Universal Robots PolyScope program: mixerHome.urp

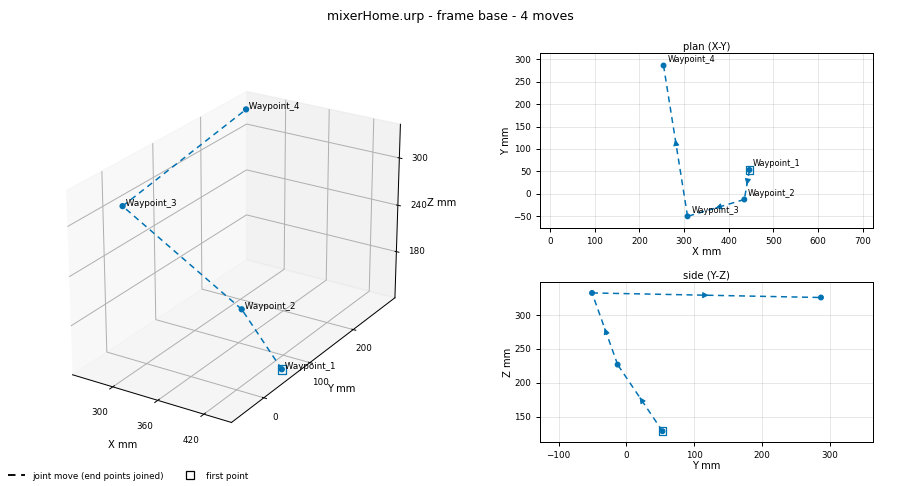
[picture p0: tool path of mixerHome.urp in frame base, 4 of 5 moves have a stored position in this frame; points joined in program order, loops and branches not executed]
Program mixerHome (installation=default directory=/programs/BaderLucas createdIn=5.12.4.1101661 lastSavedIn=5.12.4.1101661 robotSerialNumber=20225502378)
Calibrated DH parameters: a=[0.00022, -0.425328, -0.389701, 0.000059, 0.000065, 0]; d=[0.162608, 0.803456, 9.992211, -10.662202, 0.099702, 0.099559]; alpha=[1.570756, 0.001543, 0.004316, 1.570651, -1.570122, 0]; deltaTheta=[0, 0.002917, 0.116094, -0.119008, 0, -0.000001]
Robot Program (runOnlyOnce=true)
  MoveJ speed 60 deg/s, acceleration 80 deg/s^2 (useActiveTCP=true) feature=Base
    Waypoint Waypoint_1: TCP in base x=446.252 y=53.042 z=128.805 mm, rx=-0.009 ry=2.1862 rz=2.2401 rad; joints [11.497, -116.002, -118.682, -117.336, -168.067, 7.157] deg
    Waypoint Waypoint_2: TCP in base x=434.77 y=-13.057 z=226.886 mm, rx=-0.0047 ry=2.2052 rz=2.2064 rad; joints [2.918, -105.448, -113.546, -136.125, -176.254, 3.868] deg
    Waypoint Waypoint_3: TCP in base x=307.789 y=-50.757 z=332.503 mm, rx=1.5401 ry=-1.6738 rz=-1.3752 rad; joints [7.333, -85.298, -113.486, -136.131, -243.091, -5.394] deg; TCP offset x=0 y=0 z=0 mm, rx=0 ry=0 rz=0 rad
    Waypoint Waypoint_4: TCP in base x=254.1 y=286.523 z=325.774 mm, rx=2.4525 ry=-0.7929 rz=-0.5192 rad; joints [64.368, -85.38, -113.494, -104.533, -252.697, 4.851] deg; TCP offset x=0 y=0 z=0 mm, rx=0 ry=0 rz=0 rad
    Waypoint Waypoint (Variable): variable=cotonHomePos
    URCap Gripper Activate (Robotiq_Grippers, Robotiq Inc.) dataModel(ResetAndActivateKey=false)
    URCap Gripper (Robotiq_Grippers, Robotiq Inc.) dataModel(position=100.0, force=0.0, speed=0.0, positionInDouble=100.0, forceInDouble=0.0, speedInDouble=0.0, slaveIds=[9], blocking=true)
